(* CODESYS project prova1.project

Project tree, tasks and I/O mapping:
  Device : CODESYS Control Win V3, 3S - Smart Software Solutions GmbH, order no. 305021, version 3.5.11.30
    application Application
      libraries: Standard, * (System)
      task MainTask (cyclic, interval t#20ms, priority 1) calls PLC_PRG
      program PLC_PRG [LD]
*)

// Device/Application/PLC_PRG
PROGRAM PLC_PRG
VAR
	BT1: BOOL; //BOTAO LIGA SISTEMA
	TOF_0: TOF; //TEMPORIZADOR DO BATEDOR RODANDO
	KM1: BOOL; //CONTATOR QUE LIGA O MOTOR DO BATEDOR 
	TON_0: TON; //TEMPORIZADOR DO BATEDOR PARADO
	X: TIME;
	AUXTON: BOOL; //VARIAVEL AUXILIAR PARA RELIGAR O TEMPORIZADOR DA BATEDEIRA 
	BT2: BOOL; //BOTÃO QUE DESLIGA TODO O SISTEMA
	CTU_0: CTU; //CONTADOR DOS CICLOS
	TOF_1: TOF; //CONTADOR DA VALVULA
	V2: BOOL; //VALVULA
	L1: BOOL; //LAMPADA SISTEMA EM FUNCIONAMENTO
	AUX2: BOOL; //VAR AUX USADA PARA QUE O SISTEMA NAO INICIE ANTES DE APERTAR BT1
	AUX3: BOOL; //VARIAVEL AUX PARA NAO REICIAR AUTOMATICAMENETE TODO O PROCESSO APOS O SEU TERMINO
END_VAR
VAR // added by the converter: edge detectors and wires of the graphical bodies
    _w1, _w2 : BOOL;
END_VAR

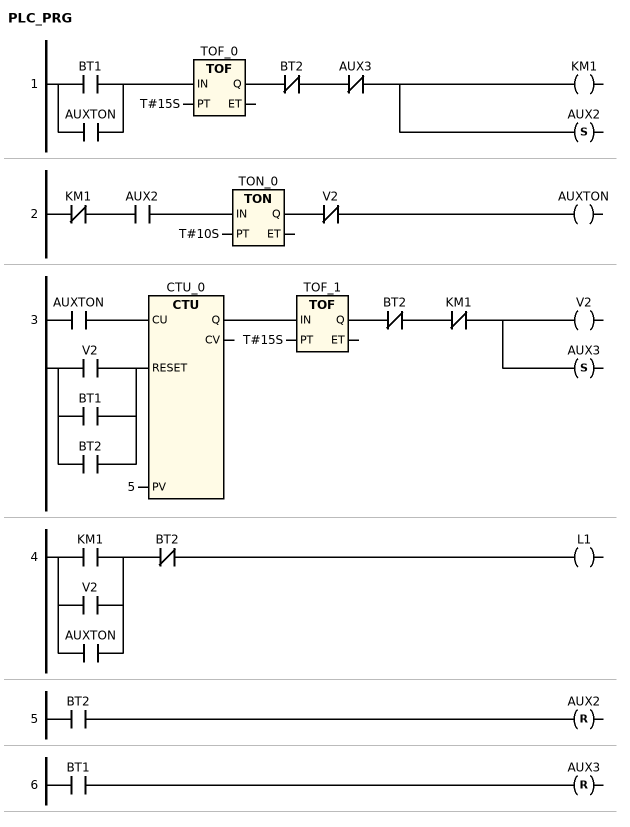
// NETWORK 1
TOF_0(IN := BT1 OR AUXTON, PT := T#15S); // TOF
_w1 := TOF_0.Q AND NOT BT2 AND NOT AUX3;
KM1 := _w1;
AUX2 S= _w1;

// NETWORK 2
TON_0(IN := NOT KM1 AND AUX2, PT := T#10S); // TON
AUXTON := TON_0.Q AND NOT V2;

// NETWORK 3
CTU_0(CU := AUXTON, RESET := V2 OR BT1 OR BT2, PV := 5); // CTU
TOF_1(IN := CTU_0.Q, PT := T#15S); // TOF
_w2 := TOF_1.Q AND NOT BT2 AND NOT KM1;
V2 := _w2;
AUX3 S= _w2;

// NETWORK 4
L1 := (KM1 OR V2 OR AUXTON) AND NOT BT2;

// NETWORK 5
AUX2 R= BT2;

// NETWORK 6
AUX3 R= BT1;

END_PROGRAM
